TYPE MFCType :
(
	MFCType_Default := 0 //常规分子MFC
)UINT;
END_TYPE

(* stored: Version 1.1.0.1, ProductVersion 3.1.4024.4
   DUT MFCType: Id {c8c6b0e6-c1d5-4b4c-9d73-e9871a771e4c} *)
